PROGRAM MAIN
VAR
	x: bool;
END_VAR

;

END_PROGRAM

(* stored: Version 1.1.0.1, ProductVersion 3.1.4024.3
   POU MAIN: Id {c0cd1fe4-1d42-4fb8-9c59-4e4085b8b27b}, SpecialFunc None *)
